FUNCTION_BLOCK FB_Derivator
VAR_INPUT
	ss_UpdateMode: SINT;
	f_Signal: LREAL;
END_VAR
VAR_OUTPUT
	f_DerivatedSignal: LREAL;
END_VAR
VAR
	rtb_TSamp: LREAL;
	UD_DSTATE: LREAL;
END_VAR

END_FUNCTION_BLOCK

(* stored: Version 1.1.0.1
   POU FB_Derivation: Id {6e2d8cc8-4fb7-48c3-b9f7-a8fc414e772e}, SpecialFunc None *)
